{attribute 'GeneratedUsingTerminal: EK1122-0000-0018'}
{attribute addProperty BoxType "EK1122-0000-0018"}
{attribute addProperty Id "Beckhoff_EJ4xxxsub_EK1100EK1100_1FC0878B2"}
{attribute addProperty CRC "3776704694"}
{attribute addProperty Size "2"}
TYPE Beckhoff_EJ4xxxEK1122_E11BF0B6 EXTENDS EK1122_1FC0878B :
STRUCT
	{attribute addProperty Name "Beckhoff EJ4xxxsub EK1100"}
	{attribute addProperty PreviousPort "Beckhoff EJ4xxxEK1122 : D"}
	Beckhoff_EJ4xxxsub_EK1100 : EK1100_1FC0878B;
END_STRUCT
END_TYPE

(* stored: Version 1.2.0.0, ProductVersion 3.1.4024.9
   DUT Beckhoff_EJ4xxxEK1122_E11BF0B6: Id {dc572d9a-8c6b-4e68-aef7-b28bdb0168fd} *)
